FUNCTION_BLOCK WriteModbusBool
VAR_INPUT
	L_Input: BOOL;
END_VAR
VAR_OUTPUT
END_VAR
VAR
	i: INT;
END_VAR


i:= GVL.nInputCoilIndex;
GVL.mb_Input_Coils[i+0]:= L_Input;

GVL.nInputCoilIndex:= i+1;

END_FUNCTION_BLOCK

(* stored: Version 1.1.0.1, ProductVersion 3.1.4024.12
   POU WriteModbusBool: Id {3206a8bd-43fb-4181-b282-68b6f0b081f4}, SpecialFunc None *)
